// TIA Portal project "FCs7-1200" (V11)

(* hardware
DEVICE "Estación SIMATIC 1200_1"  S71200.Device
   slot 0: "Rack S7-1200"  Rack  V1.0
   slot 1: "PLC_1"  CPU 1214C AC/DC/Rly  6ES7 214-1BE30-0XB0  V2.2
   slot 3: "AQ1 x 12bits_1"  6ES7 232-4HA30-0XB0  V1.0
*)

// ===== PLC "PLC_1"  CPU 1214C AC/DC/Rly =====

VAR_GLOBAL   // PLC tag table "Tabla de variables estándar"
   "Tag_1" AT %M0.0 : Bool;
   "Tag_2" AT %M0.1 : Bool;
   "System_Byte" AT %MB100 : Byte;
   "FirstScan" AT %M100.0 : Bool;
   "DiagStatusUpdate" AT %M100.1 : Bool;
   "AlwaysTRUE" AT %M100.2 : Bool;
   "AlwaysFALSE" AT %M100.3 : Bool;
   "Tag_3" AT %E0.0 : Bool;
   "Tag_4" AT %E0.1 : Bool;
   "Tag_5" AT %A0.0 : Bool;
   "Tag_6" AT %E0.2 : Bool;
   "Tag_7" AT %E0.3 : Bool;
   "Tag_8" AT %A0.1 : Bool;
   "Tag_9" AT %A0.2 : Bool;
   "Tag_10" AT %A0.3 : Bool;
   "Tag_11" AT %M0.2 : Bool;
   "Tag_12" AT %M0.4 : Bool;
   "Tag_13" AT %M0.3 : Bool;
END_VAR

DATA_BLOCK "BIT"   // DB1
{ S7_Optimized_Access := 'FALSE' }
VERSION : 0.1
   VAR
      "M0.0" : Bool;
      "M0.1" : Bool;
      "M0.2" : Bool;
      "m0.3" : Bool;
      "F0.4" : Bool;
      "F0.5" : Bool;
      "F0.6" : Bool;
      "F0.7" : Bool;
      "F0.8" : Bool;
      "M1.0" : Bool;
      "M1.1" : Bool;
      "M1.2" : Bool;
   END_VAR
BEGIN
END_DATA_BLOCK

// folder: System blocks/Program resources

DATA_BLOCK "TIM0"   // DB2
{ S7_Optimized_Access := 'FALSE' }
AUTHOR : Simatic
FAMILY : IEC
NAME : IEC_TMR
VERSION : 1.0
// stored: InstanceOfName ?
"?"
BEGIN
END_DATA_BLOCK

DATA_BLOCK "TIM1"   // DB3
{ S7_Optimized_Access := 'FALSE' }
AUTHOR : Simatic
FAMILY : IEC
NAME : IEC_TMR
VERSION : 1.0
// stored: InstanceOfName ?
"?"
BEGIN
END_DATA_BLOCK

DATA_BLOCK "TIM2"   // DB4
{ S7_Optimized_Access := 'FALSE' }
AUTHOR : Simatic
FAMILY : IEC
NAME : IEC_TMR
VERSION : 1.0
// stored: InstanceOfName ?
"?"
BEGIN
END_DATA_BLOCK

// folder: (top level)

FUNCTION "FC 1 ARRANQUE DIRECTO" : Void   // FC1, LAD
{ S7_Optimized_Access := 'FALSE' }
VERSION : 0.1
   VAR_INPUT
      MARCHA : Bool;
      PARO : Bool;
   END_VAR
   VAR_OUTPUT
      MOTOR : Bool;
   END_VAR
BEGIN

REGION Network 1
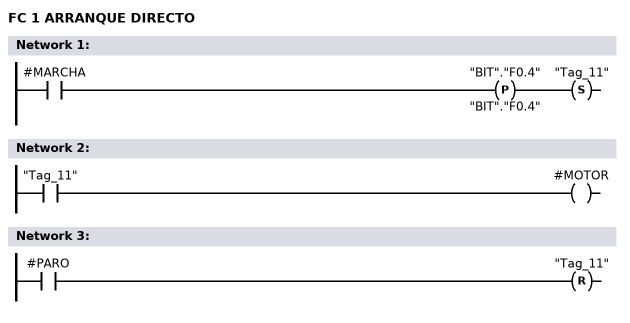
   "BIT"."F0.4" := #MARCHA AND NOT "BIT"."F0.4";   // rising edge
   "BIT"."F0.4" := #MARCHA;
   IF #MARCHA THEN "Tag_11" := TRUE; END_IF;
END_REGION

REGION Network 2
   RUNG wire#powerrail
      Contact( "Tag_11" )
      Coil( #MOTOR )
   END_RUNG
   // the same network as SCL:
   #MOTOR := "Tag_11";
END_REGION

REGION Network 3
   RUNG wire#powerrail
      Contact( #PARO )
      R_Coil( "Tag_11" )
   END_RUNG
   // the same network as SCL:
   IF #PARO THEN "Tag_11" := FALSE; END_IF;
END_REGION
END_FUNCTION

FUNCTION "FC 2 ESTRELLA-TRIANGULO" : Void   // FC2, LAD
{ S7_Optimized_Access := 'FALSE' }
VERSION : 0.1
   VAR_INPUT
      MARCHA : Bool;
      PARO : Bool;
   END_VAR
   VAR_OUTPUT
      LINEA : Bool;
      ESTRELLA : Bool;
      TRIANGULO : Bool;
   END_VAR
   VAR_TEMP   // added for the SCL form of the ladder/FBD networks
      _w1 : Bool;
   END_VAR
BEGIN

REGION Network 1
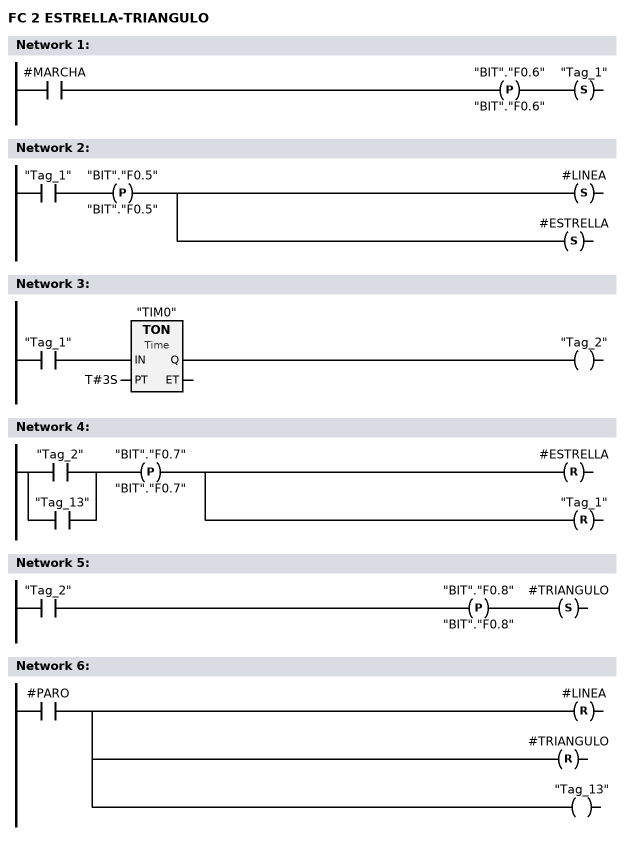
   "BIT"."F0.6" := #MARCHA AND NOT "BIT"."F0.6";   // rising edge
   "BIT"."F0.6" := #MARCHA;
   IF #MARCHA THEN "Tag_1" := TRUE; END_IF;
END_REGION

REGION Network 2
   "BIT"."F0.5" := "Tag_1" AND NOT "BIT"."F0.5";   // rising edge
   "BIT"."F0.5" := "Tag_1";
   IF "Tag_1" THEN
       #LINEA := TRUE;
       #ESTRELLA := TRUE;
   END_IF;
END_REGION

REGION Network 3
   "TIM0".TON(IN := "Tag_1", PT := T#3S);
   "Tag_2" := "TIM0".Q;
END_REGION

REGION Network 4
   #_w1 := "Tag_2" OR "Tag_13";
   "BIT"."F0.7" := #_w1 AND NOT "BIT"."F0.7";   // rising edge
   "BIT"."F0.7" := #_w1;
   IF #_w1 THEN
       #ESTRELLA := FALSE;
       "Tag_1" := FALSE;
   END_IF;
END_REGION

REGION Network 5
   "BIT"."F0.8" := "Tag_2" AND NOT "BIT"."F0.8";   // rising edge
   "BIT"."F0.8" := "Tag_2";
   IF "Tag_2" THEN #TRIANGULO := TRUE; END_IF;
END_REGION

REGION Network 6
   RUNG wire#powerrail
      Contact( #PARO )
      wire#w1
      R_Coil( #LINEA )
   END_RUNG
   RUNG wire#w1
      R_Coil( #TRIANGULO )
   END_RUNG
   RUNG wire#w1
      Coil( "Tag_13" )
   END_RUNG
   // the same network as SCL:
   IF #PARO THEN
       #LINEA := FALSE;
       #TRIANGULO := FALSE;
   END_IF;
   "Tag_13" := #PARO;
END_REGION
END_FUNCTION

ORGANIZATION_BLOCK "Main"   // OB1, LAD, ProgramCycle
TITLE = "Main Program Sweep (Cycle)"
{ S7_Optimized_Access := 'FALSE' }
VERSION : 0.1
BEGIN

REGION Network 1
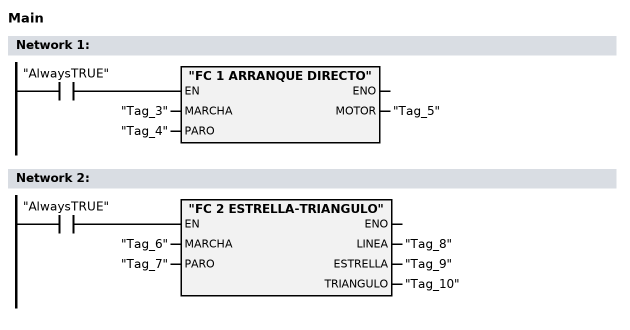
   RUNG wire#powerrail
      Contact( "AlwaysTRUE" )
      "FC 1 ARRANQUE DIRECTO"(MARCHA := "Tag_3", PARO := "Tag_4", MOTOR => "Tag_5")
   END_RUNG
   // the same network as SCL:
   IF "AlwaysTRUE" THEN
       "FC 1 ARRANQUE DIRECTO"(MARCHA := "Tag_3", PARO := "Tag_4", MOTOR => "Tag_5");
   END_IF;
END_REGION

REGION Network 2
   RUNG wire#powerrail
      Contact( "AlwaysTRUE" )
      "FC 2 ESTRELLA-TRIANGULO"(MARCHA := "Tag_6", PARO := "Tag_7", LINEA => "Tag_8", ESTRELLA => "Tag_9", TRIANGULO => "Tag_10")
   END_RUNG
   // the same network as SCL:
   IF "AlwaysTRUE" THEN
       "FC 2 ESTRELLA-TRIANGULO"(MARCHA := "Tag_6",
                               PARO := "Tag_7",
                               LINEA => "Tag_8",
                               ESTRELLA => "Tag_9",
                               TRIANGULO => "Tag_10");
   END_IF;
END_REGION
END_ORGANIZATION_BLOCK

// ===== library: MasterCopy "Copia de PLC_1" =====

ORGANIZATION_BLOCK "Main"   // OB1, LAD, ProgramCycle
TITLE = "Main Program Sweep (Cycle)"
{ S7_Optimized_Access := 'FALSE' }
VERSION : 0.1
BEGIN
END_ORGANIZATION_BLOCK